PROGRAM P00_Mapping
VAR
END_VAR

END_PROGRAM

(* stored: Version 1.1.0.1
   POU P00_Mapping: Id {a71a5ccb-5f7c-4f94-87c7-70455710a762}, SpecialFunc None *)
